// TIA Portal V19 export
TYPE "udt_MbClient"
// stored: Access Published
   STRUCT
      req : Bool;   // Activates the requested transmission if TRUE
      disconnect : Bool;   // Initiates a disconnect operation
      mode : USInt;   // Specifies the type of request: read, write or diagnostic
      DataAddr : UDInt;   // Specifies the starting address of the data to be accessed in the Modbus client
      DataLen : UInt;
      connect { S7_SetPoint := 'True'} : TCON_IP_v4;   // Reference to the connection parameters
   END_STRUCT;
   // connect.InterfaceId := 64;
   // connect.ID := 1;
   // connect.ActiveEstablished := true;
   // connect.RemoteAddress.ADDR[1] := 192;
   // connect.RemoteAddress.ADDR[2] := 168;
   // connect.RemoteAddress.ADDR[3] := 0;
   // connect.RemotePort := 502;
END_TYPE
